Omron CX-Programmer project NewProject (CX-Programmer 9.61)

# PLC Parfum_Otomatis: CP1L L

## Global symbols (name address type ; comment)
100.13 BOOL  ; Valve
10.10 BOOL  ; IR Stop
10.05 BOOL  ; Running 2
100.12 BOOL  ; Botol Packing
0.05 BOOL  ; Sensor Pelabelan
0.04 BOOL  ; Sensor Botol
100.14 BOOL  ; Botol Packing
100.04 BOOL  ; Motor Pengaduk
0.06 BOOL  ; Sensor Proximity
10.00 BOOL  ; Running 1
0.00 BOOL  ; Start
0.01 BOOL  ; Stop
0.02 BOOL  ; Emergency
0.07 BOOL  ; Sensor Proximity
0.08 BOOL  ; Counter Reset
100.00 BOOL  ; Pompa 1
100.01 BOOL  ; Pompa 1
100.02 BOOL  ; Pompa 2
100.03 BOOL  ; Pompa 3
100.05 BOOL  ; Conveyor 1
100.06 BOOL  ; Isi Botol
100.07 BOOL  ; Tutup Botol
100.08 BOOL  ; Conveyor 2
100.09 BOOL  ; Conveyor 3
100.10 BOOL  ; Pelabelan
100.11 BOOL  ; Packing
100.15 BOOL  ; IR RUN 2
10.01 BOOL  ; Max Athyl Alcohol
10.02 BOOL  ; Max Aqua
10.03 BOOL  ; Max Pewangi
10.04 BOOL  ; Max Keselutuhan
10.06 BOOL  ; Min Athyl Alcohol
10.07 BOOL  ; Min Aqua
10.08 BOOL  ; Min Pewangi
10.09 BOOL  ; Min Keseluruhan
10.11 BOOL  ; Pelabelan
10.12 BOOL  ; Coneyor 3
10.13 BOOL  ; Running 2
C0000 BOOL  ; Counter Packing
T0000 BOOL  ; Timer Pengaduk
T0001 BOOL  ; Timer Conv 2
T0002 BOOL  ; Timer Isi
T0003 BOOL  ; Timer Tutup
T0004 BOOL  ; Timer Conv
T0005 BOOL  ; Timer Pelabelan
T0006 BOOL  ; Timer Conveyor 2
T0007 BOOL  ; Counter Reset

## Program NewProgram1 (cyclic task 0)
Local symbols
Running BOOL

### Section Section1

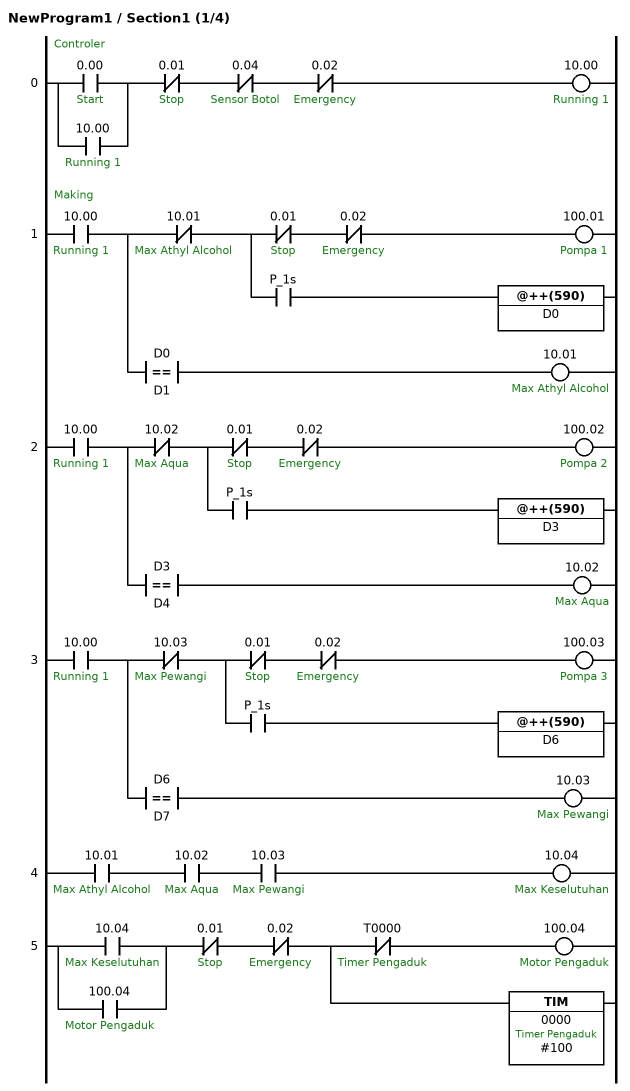
; rung 0: Controler
LD 0.00  ; Start
OR 10.00  ; Running 1
ANDNOT 0.01  ; Stop
ANDNOT 0.04  ; Sensor Botol
ANDNOT 0.02  ; Emergency
OUT 10.00  ; Running 1
; rung 1: Making
LD 10.00  ; Running 1
OUT TR0
ANDNOT 10.01  ; Max Athyl Alcohol
OUT TR1
ANDNOT 0.01  ; Stop
ANDNOT 0.02  ; Emergency
OUT 100.01  ; Pompa 1
LD TR1
AND P_1s
@++(590) D0
LD TR0
AND=(300) D0 D1
OUT 10.01  ; Max Athyl Alcohol
; rung 2
LD 10.00  ; Running 1
OUT TR0
ANDNOT 10.02  ; Max Aqua
OUT TR1
ANDNOT 0.01  ; Stop
ANDNOT 0.02  ; Emergency
OUT 100.02  ; Pompa 2
LD TR1
AND P_1s
@++(590) D3
LD TR0
AND=(300) D3 D4
OUT 10.02  ; Max Aqua
; rung 3
LD 10.00  ; Running 1
OUT TR0
ANDNOT 10.03  ; Max Pewangi
OUT TR1
ANDNOT 0.01  ; Stop
ANDNOT 0.02  ; Emergency
OUT 100.03  ; Pompa 3
LD TR1
AND P_1s
@++(590) D6
LD TR0
AND=(300) D6 D7
OUT 10.03  ; Max Pewangi
; rung 4
LD 10.01  ; Max Athyl Alcohol
AND 10.02  ; Max Aqua
AND 10.03  ; Max Pewangi
OUT 10.04  ; Max Keselutuhan
; rung 5
LD 10.04  ; Max Keselutuhan
OR 100.04  ; Motor Pengaduk
ANDNOT 0.01  ; Stop
ANDNOT 0.02  ; Emergency
OUT TR0
ANDNOT T0000  ; Timer Pengaduk
OUT 100.04  ; Motor Pengaduk
LD TR0
TIM 0000 #100  ; Timer Pengaduk

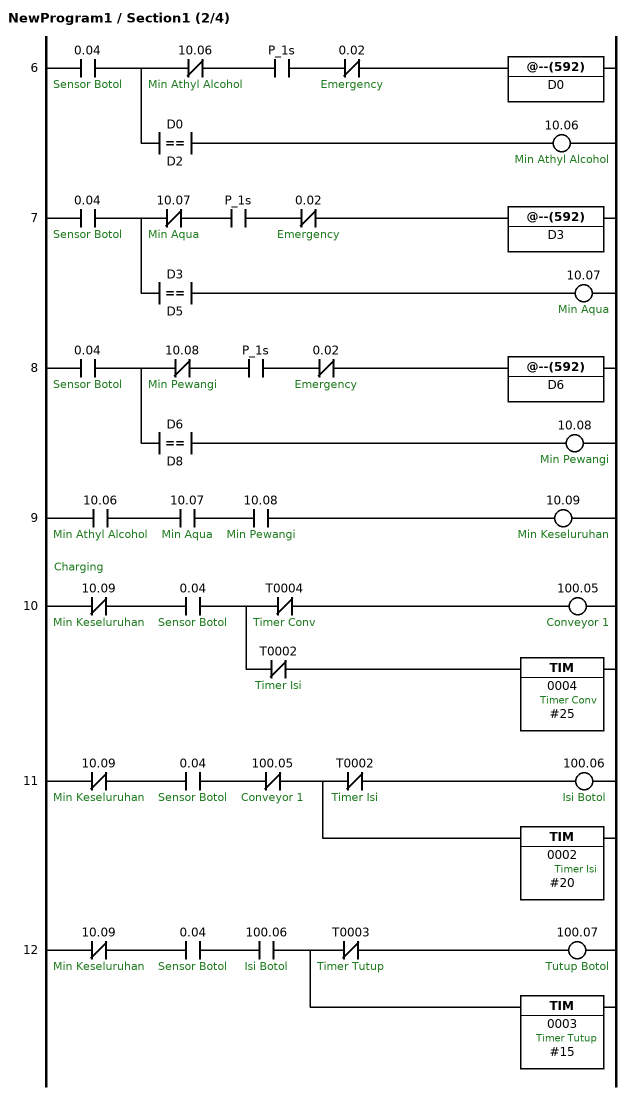
; rung 6
LD 0.04  ; Sensor Botol
OUT TR0
ANDNOT 10.06  ; Min Athyl Alcohol
AND P_1s
ANDNOT 0.02  ; Emergency
@--(592) D0
LD TR0
AND=(300) D0 D2
OUT 10.06  ; Min Athyl Alcohol
; rung 7
LD 0.04  ; Sensor Botol
OUT TR0
ANDNOT 10.07  ; Min Aqua
AND P_1s
ANDNOT 0.02  ; Emergency
@--(592) D3
LD TR0
AND=(300) D3 D5
OUT 10.07  ; Min Aqua
; rung 8
LD 0.04  ; Sensor Botol
OUT TR0
ANDNOT 10.08  ; Min Pewangi
AND P_1s
ANDNOT 0.02  ; Emergency
@--(592) D6
LD TR0
AND=(300) D6 D8
OUT 10.08  ; Min Pewangi
; rung 9
LD 10.06  ; Min Athyl Alcohol
AND 10.07  ; Min Aqua
AND 10.08  ; Min Pewangi
OUT 10.09  ; Min Keseluruhan
; rung 10: Charging
LDNOT 10.09  ; Min Keseluruhan
AND 0.04  ; Sensor Botol
OUT TR0
ANDNOT T0004  ; Timer Conv
OUT 100.05  ; Conveyor 1
LD TR0
ANDNOT T0002  ; Timer Isi
TIM 0004 #25  ; Timer Conv
; rung 11
LDNOT 10.09  ; Min Keseluruhan
AND 0.04  ; Sensor Botol
ANDNOT 100.05  ; Conveyor 1
OUT TR0
ANDNOT T0002  ; Timer Isi
OUT 100.06  ; Isi Botol
LD TR0
TIM 0002 #20  ; Timer Isi
; rung 12
LDNOT 10.09  ; Min Keseluruhan
AND 0.04  ; Sensor Botol
AND 100.06  ; Isi Botol
OUT TR0
ANDNOT T0003  ; Timer Tutup
OUT 100.07  ; Tutup Botol
LD TR0
TIM 0003 #15  ; Timer Tutup

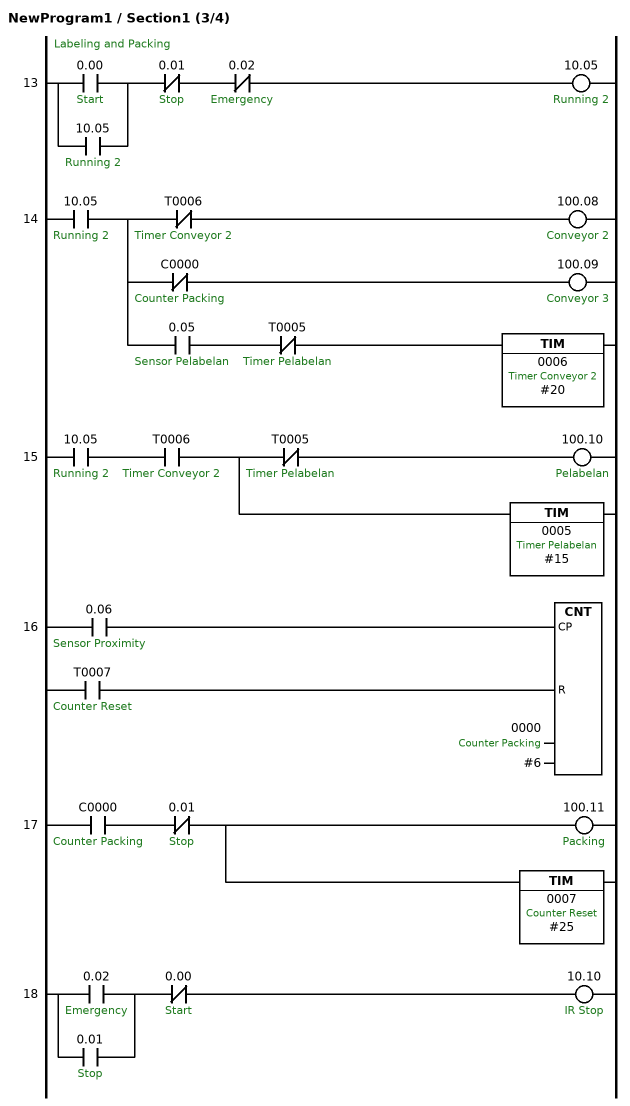
; rung 13: Labeling and Packing
LD 0.00  ; Start
OR 10.05  ; Running 2
ANDNOT 0.01  ; Stop
ANDNOT 0.02  ; Emergency
OUT 10.05  ; Running 2
; rung 14
LD 10.05  ; Running 2
OUT TR0
ANDNOT T0006  ; Timer Conveyor 2
OUT 100.08  ; Conveyor 2
LD TR0
ANDNOT C0000  ; Counter Packing
OUT 100.09  ; Conveyor 3
LD TR0
AND 0.05  ; Sensor Pelabelan
ANDNOT T0005  ; Timer Pelabelan
TIM 0006 #20  ; Timer Conveyor 2
; rung 15
LD 10.05  ; Running 2
AND T0006  ; Timer Conveyor 2
OUT TR0
ANDNOT T0005  ; Timer Pelabelan
OUT 100.10  ; Pelabelan
LD TR0
TIM 0005 #15  ; Timer Pelabelan
; rung 16
LD 0.06  ; Sensor Proximity
LD T0007  ; Counter Reset
CNT 0000 #6  ; Counter Packing
; rung 17
LD C0000  ; Counter Packing
ANDNOT 0.01  ; Stop
OUT 100.11  ; Packing
TIM 0007 #25  ; Counter Reset
; rung 18
LD 0.02  ; Emergency
OR 0.01  ; Stop
ANDNOT 0.00  ; Start
OUT 10.10  ; IR Stop

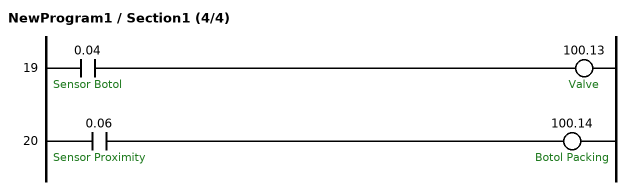
; rung 19
LD 0.04  ; Sensor Botol
OUT 100.13  ; Valve
; rung 20
LD 0.06  ; Sensor Proximity
OUT 100.14  ; Botol Packing
; rung 21
END(001)

### Section END
; rung 0
END(001)